FUNCTION_BLOCK ESP32_Testboard_8_DI_DOUBLE_CLICK (* Service Interface Function Block Type *)
  (* Function: All Inputs; Description: this maps to IE *)
  (* Version 1.0, 2018-12-05, Jose Cabral *)
  (* Version 1.1, 2022-08-04, Franz Höpfinger, HR Agrartechnik GmbH *)
  (* Version 1.2, 2023-01-05, Franz Höpfinger, HR Agrartechnik GmbH *)
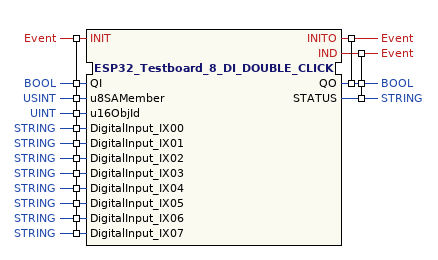
  EVENT_INPUT
    INIT WITH QI, u8SAMember, u16ObjId, DigitalInput_IX00, DigitalInput_IX01, DigitalInput_IX02, DigitalInput_IX03, DigitalInput_IX04, DigitalInput_IX05, DigitalInput_IX06, DigitalInput_IX07; (* Service Initialization *)
  END_EVENT
  EVENT_OUTPUT
    INITO WITH QO; (* Initialization Confirm *)
    IND WITH QO, STATUS; (* Indication from Resource *)
  END_EVENT
  VAR_INPUT
    QI : BOOL; (* Event Input Qualifier *)
    u8SAMember : USINT := GLOBAL; (* Dummy !, set to GLOBAL if in doubt. OFF deactivates FB. *)
    u16ObjId : UINT := ID_NULL; (* Dummy ! set to ID_NULL if in Doubt. ID_OFF deactivates FB. *)
    DigitalInput_IX00 : STRING; (* Identifier for Input 0 *)
    DigitalInput_IX01 : STRING; (* Identifier for Input 1 *)
    DigitalInput_IX02 : STRING; (* Identifier for Input 2 *)
    DigitalInput_IX03 : STRING; (* Identifier for Input 3 *)
    DigitalInput_IX04 : STRING; (* Identifier for Input 4 *)
    DigitalInput_IX05 : STRING; (* Identifier for Input 5 *)
    DigitalInput_IX06 : STRING; (* Identifier for Input 6 *)
    DigitalInput_IX07 : STRING; (* Identifier for Input 7 *)
  END_VAR
  VAR_OUTPUT
    QO : BOOL; (* Event Output Qualifier *)
    STATUS : STRING; (* Service Status *)
  END_VAR
END_FUNCTION_BLOCK
